{attribute 'GeneratedUsingTerminal: KL2819'}
{attribute addProperty BoxType "KL2819"}
{attribute addProperty Id "StatusAT %I*USINT0DiagAT %I*WORD0CtrlAT %Q*USINT0OutputAT %Q*WORD0"}
{attribute addProperty CRC "784591050"}
{attribute addProperty Size "0"}
TYPE Channel_2EC3E8CA :
STRUCT
	{attribute addProperty Name "Status"}
	Status AT %I* : USINT;
	{attribute addProperty Name "Diag"}
	Diag AT %I* : WORD;
	{attribute addProperty Name "Ctrl"}
	Ctrl AT %Q* : USINT;
	{attribute addProperty Name "Output"}
	Output AT %Q* : WORD;
END_STRUCT
END_TYPE

(* stored: Version 1.2.0.0, ProductVersion 3.1.4024.9
   DUT Channel_2EC3E8CA: Id {42781de4-68a2-4e28-948c-87197b0e31d2} *)
